# EPICS alarm handler configuration: mps_database/bareTest/alarms/areas/mpln_unds_mp01.alhConfig
GROUP NULL MPLN:UNDS:MP01:1
$ALIAS MPS Link Node 208
$GUIDANCE
LTUH MPS
   Group Name: MPLN:UNDS:MP01:1
   Summary PV:  MPLN:UNDS:MP01:1:STATSUMY
$END
CHANNEL  MPLN:UNDS:MP01:1    MPLN:UNDS:MP01:1:MPS_EN_RBV		-----
CHANNEL  MPLN:UNDS:MP01:1    MPLN:UNDS:MP01:1:LC1_MODE_RBV		-----
